(* Logix 5000 project; controller Receptivo vendor 1 type 14 code 106 rev 30.11; software revision 30.00; part 3 of 10 *)

   Impreso_3 : BOOL;
   Impreso_4 : BOOL;
   Imprimiendo_1 : BOOL;
   Imprimiendo_1_Timer : TIMER := (PRE := 7000);
   Imprimiendo_2 : BOOL;
   Imprimiendo_2_Timer : TIMER := (PRE := 7000);
   Imprimiendo_3 : BOOL;
   Imprimiendo_3_Timer : TIMER := (PRE := 7000);
   Imprimiendo_4 : BOOL;
   Imprimiendo_4_Timer : TIMER := (PRE := 7000);
   Index_Bidones_Videojet : DINT;
   Index_Elmar_Videojet : DINT := 112;
   Index_Fogg1_Videojet : DINT := 203;
   Index_Fogg2_Videojet : DINT := 23;
   Index_Karat_Videojet : DINT;
   Index_Karat_Videojet_Antiguo : DINT;
   Index_Productos : DINT := 118;
   Index_S : INT := 200;
   Index_Scanner : COUNTER := (PRE := 300, ACC := 3483, DN := 1);
   Indice_Bidon_Videojet : DINT;
   KEY_SWITCH_REM_RUN : BOOL := 1;
   KEY_SWITCH_RUN : BOOL;
   Latch_Scanner_1 : BOOL := 1;
   Latch_Scanner_2 : BOOL;
   Latch_Scanner_3 : BOOL;
   Lectura_Efectuada : BOOL;
   Linea_1 : SINT;
   Linea_2 : SINT;
   Linea_3 : SINT;
   Linea_4 : SINT;
   Linea_5 : SINT;
   Linea_General : SINT;
   LInea_General_1 : INT := 3;
   LInea_General_2 : INT := 1;
   LInea_General_3 : INT := 3;
   LInea_General_4 : INT := 5;
   Linea_String_General : STRING := '5';
   Listado : INT := 9;
   Listado_A : INT := 9;
   Lote : DINT := 148;
   Mes_dias : INT[13] := ([2] := 31, [3] := 59, [4] := 90, [5] := 120, [6] := 151, [7] := 181, [8] := 212, [9] := 243, [10] := 273, [11] := 304, [12] := 334);
   MODULE_FAULT_STATUS : DINT[10];
   Modulo_Ethernet_Mal : BOOL;
   new_day : BOOL;
   No_CAJAS_1 : DINT;
   No_CAJAS_2 : DINT;
   No_CAJAS_3 : DINT;
   No_existe : Descripcion := 'Codigo No Existe En El Inventario';
   Nuevo_Lote_Fogg1 : BOOL;
   Num_Cajas_Reales_1 : DINT;
   Num_Cajas_Reales_2 : DINT;
   Num_Cajas_Reales_3 : DINT;
   Num_Cajas_Reales_4 : DINT;
   Numero_Datos : DINT := 300;
   ons_add : BOOL;
   ons_add2 : BOOL;
   ons_add3 : BOOL;
   ons_add4 : BOOL;
   Ons_Cola2 : BOOL;
   Ons_Cola3 : BOOL;
   Ons_Corte_Dia : BOOL;
   ons_datos_mal_Bidones : BOOL;
   ons_datos_mal_elmar : BOOL;
   ons_datos_mal_Fogg1 : BOOL;
   ons_datos_mal_Fogg2 : BOOL;
   Ons_Datos_Mal_Karat : BOOL;
   ons_densidad_elmar : BOOL;
   ons_densidad_Fogg_1 : BOOL;
   Ons_Densidad_Karat : BOOL;
   Ons_NP : BOOL;
   Ons_NP2 : BOOL;
   Ons_NP3 : BOOL;
   Ons_NP4 : BOOL;
   Ons_Nuevo_Karat_Videojet : BOOL;
   ons_peso_caja_elmar_2 : BOOL;
   ONS_Reporte_Dia : BOOL;
   ons_scanner_1 : BOOL := 1;
   ons_scanner_3 : BOOL;
   ons_tare_station_4 : BOOL;
   Operador_1 : DINT := 5;
   Operador_2 : DINT := 5;
   Operador_3 : DINT := 5;
   Operador_4 : DINT := 6;
   PB_Enable_Scanner_1 : BOOL := 1;
   PB_Enable_Scanner_2 : BOOL;
   PB_Enable_Scanner_3 : BOOL;
   PB_Pesaje_1 : BOOL;
   PB_PV_Entre_Peso_Caja_Elmar : BOOL;
   PB_Tare_Station_1 : BOOL;
   PB_Tare_Station_2 : BOOL;
   PB_Tare_Station_3 : BOOL;
   PB_Tare_Station_4 : BOOL;
   Pesaje_1 : REAL := 0.6;
   Pesaje_2 : REAL := 0.6;
   Pesaje_3 : REAL := 0.9;
   Pesaje_4 : REAL := 0.102;
   Pesaje_Elmar_OK : BOOL;
   Pesaje_Fogg1_OK : BOOL;
   Pesaje_Fogg2_OK : BOOL;
   Pesaje_Karat_OK : BOOL;
   Peso_Aux : DINT;
   Peso_Aux_Scanner : STRING;
   Peso_Bidon : REAL;
   Peso_Bidones : REAL;
   Peso_Bidones_1 : REAL := 0.102;
   Peso_Caja_Bidones : REAL;
   Peso_Caja_Bidones_1 : REAL;
   Peso_Caja_Elmar : REAL;
   Peso_Caja_Elmar_1 : REAL := 0.6;
   Peso_Caja_Fogg1 : REAL;
   Peso_Caja_Fogg1_1 : REAL := 1.0;
   Peso_Caja_Fogg2 : REAL;
   Peso_Caja_Fogg2_1 : REAL := 0.9;
   Peso_Caja_Karat : REAL;
   Peso_Caja_Karat_1 : REAL;
   Peso_Mal_Estacion_1 : BOOL;
   Peso_Mal_Estacion_2 : BOOL;
   Peso_OK_Estacion_1 : BOOL;
   Peso_OK_Estacion_2 : BOOL;
   Peso_OK_Estacion_3 : BOOL;
   Peso_OK_Estacion_4 : BOOL;
   PESO_REAL_1 : DINT := -23;
   PESO_REAL_2 : DINT := -30;
   PESO_REAL_3 : DINT;
   PESO_REAL_4 : DINT := -23;
   PESO_TEORICO_1 : DINT := 865;
   PESO_TEORICO_2 : DINT := 585;
   PESO_TEORICO_3 : DINT := 865;
   PESO_TEORICO_4 : DINT := 786;
   Porcentaje_Peso_1 : REAL := 12257.143;
   Porcentaje_Peso_2 : REAL := 8257.143;
   Porcentaje_Peso_21 : DINT := 100;
   Porcentaje_Peso_3 : REAL := 10712.5;
   Porcentaje_Peso_4 : REAL := 1865.0;
   Print_1 : BOOL;
   Print_2 : BOOL;
   Print_3 : BOOL;
   Print_4 : BOOL;
   Printing_Enable : BOOL := 1;
   Producido_Bidones_Ahora : UDT_Maestro := (Descripcion := 'Dotchi Bidon x 20 L');
   Producido_Elmar_Ahora : UDT_Maestro := (Peso_Real_Estiba := 703.44, Peso_Teorico_Caja := 10.45, Codigo_EAN := '17702161409646', Codigo_QAD := '600620', Codigo_GCO := 600620, Descripcion := 'Alegria Caja 12 x 900 cm3  - Costa', Cajas_X_Estiba := 56, Codigo_Aceite := 600620, Envase := 900, Envases_x_Caja := 12);
   Producido_Fogg1_Ahora : UDT_Maestro := (Peso_Real_Estiba := 869.0, Peso_Teorico_Caja := 17.48, Codigo_EAN := '27702179003208', Codigo_QAD := '607490', Codigo_GCO := 607490, Descripcion := 'Vivi FF Caja 9 x2000 cm3 ', Cajas_X_Estiba := 42, Clima := 2, Codigo_Aceite := 607490, Envase := 2000, Envases_x_Caja := 9);
   Producido_Fogg2_Ahora : UDT_Maestro := (Peso_Real_Estiba := 691.2, Peso_Teorico_Caja := 17.3, Codigo_EAN := '17702161567070', Codigo_QAD := '605990', Codigo_GCO := 605990, Descripcion := 'Oriental 100% oleina x 3000 ML  Cj 6 Und', Cajas_X_Estiba := 50, Codigo_Aceite := 605990, Envase := 3000, Envases_x_Caja := 6);
   Producido_Karat_Ahora : UDT_Maestro;
   Producto1 : UDT_Inventario := (Peso_Teorico_Caja := 17.3, Descripcion := 'Oriental 100% ole$EDna x 3000 ML  Cj 6 Und', CajaXEstiba := 50, Codigo_Aceite := -1);
   Producto2 : UDT_Inventario := (Peso_Teorico_Caja := 10.45, Descripcion := 'Alegria Caja 12 x 900 cm3  - Costa', CajaXEstiba := 56, Codigo_Aceite := -1);
   Producto3 : UDT_Inventario := (Peso_Teorico_Caja := 17.3, Descripcion := 'Oriental 100% oleina x 3000 ML  Cj 6 Und', CajaXEstiba := 50, Codigo_Aceite := -1);
   Producto4 : UDT_Inventario := (Peso_Teorico_Caja := 16.38, Descripcion := 'Aceite Vegetal Torino  Exp.', CajaXEstiba := 48, Codigo_Aceite := -1);
   Producto_Codigo_Aceite_1 : DINT := -1;
   Producto_Codigo_Aceite_2 : DINT := -1;
   Producto_Codigo_Aceite_3 : DINT := -1;
   Producto_Codigo_Aceite_4 : DINT := -1;
   Producto_Scanner_1 : UDT_QAD;
   Producto_Scanner_11 : UDT_EAN14;
   Productos : UDT_Maestro[300] := ([0].Peso_Real_Estiba := 634.88, [0].Peso_Teorico_Caja := 14.72, [0].Codigo_EAN := '77702161305087', [0].Codigo_QAD := '600130', [0].Codigo_GCO := 600130, [0].Descripcion := 'Alegria Bidon x 15 L', [0].Cajas_X_Estiba := 48, [0].Clima := 2, [0].Codigo_Aceite := 600130, [0].Envase := 15000, [0].Envases_x_Caja := 1, [1].Peso_Real_Estiba := 690.84, [1].Peso_Teorico_Caja := 18.95, [1].Codigo_EAN := '07702161500506', [1].Codigo_QAD := '600100', [1].Codigo_GCO := 600100, [1].Descripcion := 'Alegria Bidon x 20 L', [1].Cajas_X_Estiba := 48, [1].Clima := 2, [1].Codigo_Aceite := 600100, [1].Envase := 20000, [1].Envases_x_Caja := 1, [2].Peso_Real_Estiba := 731.5, [2].Peso_Teorico_Caja := 18.8, [2].Codigo_EAN := '17702161574078', [2].Codigo_QAD := '606890', [2].Codigo_GCO := 606890, [2].Descripcion := 'Vivi FF Bidon x 20 L ', [2].Cajas_X_Estiba := 48, [2].Clima := 2, [2].Codigo_Aceite := 606890, [2].Envase := 20000, [2].Envases_x_Caja := 1, [3].Peso_Real_Estiba := 622.56, [3].Peso_Teorico_Caja := 19.31, [3].Codigo_EAN := '17702161071010', [3].Codigo_QAD := '606980', [3].Codigo_GCO := 606980, [3].Descripcion := 'Vivi FF Caja 4 x 5000 cm3 ', [3].Cajas_X_Estiba := 36, [3].Clima := 2, [3].Codigo_Aceite := 606980, [3].Envase := 5000, [3].Envases_x_Caja := 4, [4].Peso_Real_Estiba := 878.0, [4].Peso_Teorico_Caja := 17.4, [4].Codigo_EAN := '17702161987403', [4].Codigo_QAD := '607280', [4].Codigo_GCO := 607280, [4].Descripcion := 'Vivi FF Caja 6 x 3000 cm3 ', [4].Cajas_X_Estiba := 50, [4].Clima := 2, [4].Codigo_Aceite := 607280, [4].Envase := 3000, [4].Envases_x_Caja := 6, [5].Peso_Real_Estiba := 636.24, [5].Peso_Teorico_Caja := 17.54, [5].Codigo_EAN := '17702161845956', [5].Codigo_QAD := '607490', [5].Codigo_GCO := 607490,
        [5].Descripcion := 'Vivi FF Caja 9 x2000 cm3 ', [5].Cajas_X_Estiba := 42, [5].Clima := 2, [5].Codigo_Aceite := 607490, [5].Envase := 2000, [5].Envases_x_Caja := 9, [6].Peso_Real_Estiba := 627.2, [6].Peso_Teorico_Caja := 11.69, [6].Codigo_EAN := '17702161585364', [6].Codigo_QAD := '607690', [6].Codigo_GCO := 607690, [6].Descripcion := 'Vivi FF Caja 12 x 1000 cm3 ', [6].Cajas_X_Estiba := 70, [6].Clima := 2, [6].Codigo_Aceite := 607690, [6].Envase := 1000, [6].Envases_x_Caja := 12, [7].Peso_Real_Estiba := 830.0, [7].Peso_Teorico_Caja := 10.57, [7].Codigo_EAN := '17702161701764', [7].Codigo_QAD := '607890', [7].Codigo_GCO := 607890, [7].Descripcion := 'Vivi FF Caja 12 x 900 cm3 ', [7].Cajas_X_Estiba := 70, [7].Clima := 2, [7].Codigo_Aceite := 607890, [7].Envase := 900, [7].Envases_x_Caja := 12, [8].Peso_Real_Estiba := 625.1, [8].Peso_Teorico_Caja := 11.79, [8].Codigo_EAN := '17702161377068', [8].Codigo_QAD := '608090', [8].Codigo_GCO := 608090, [8].Descripcion := 'Vivi FF Caja 24 x 500 cm3 ', [8].Cajas_X_Estiba := 70, [8].Clima := 2, [8].Codigo_Aceite := 608090, [8].Envase := 500, [8].Envases_x_Caja := 24, [9].Peso_Real_Estiba := 770.0, [9].Peso_Teorico_Caja := 6.06, [9].Codigo_EAN := '17702161560002', [9].Codigo_QAD := '608290', [9].Codigo_GCO := 608290, [9].Descripcion := 'Vivi FF Caja 24 x 250 cm3 ', [9].Cajas_X_Estiba := 104, [9].Clima := 2, [9].Codigo_Aceite := 608290, [9].Envase := 250, [9].Envases_x_Caja := 24, [10].Peso_Real_Estiba := 883.2, [10].Peso_Teorico_Caja := 15.32, [10].Codigo_EAN := '67702179051603', [10].Codigo_QAD := '606280', [10].Codigo_GCO := 606280, [10].Descripcion := 'Comisariato Grasco Caja 6 x 2625 cm3', [10].Cajas_X_Estiba := 50, [10].Clima := 2, [10].Codigo_Aceite := 606280, [10].Envase := 2625,
        [10].Envases_x_Caja := 6, [11].Peso_Real_Estiba := 819.0, [11].Peso_Teorico_Caja := 17.27, [11].Codigo_EAN := '11111111111111', [11].Codigo_QAD := '602800', [11].Codigo_GCO := 602800, [11].Descripcion := 'La Muneca Comisariato Caja 6 x 3000 cm3', [11].Cajas_X_Estiba := 20, [11].Codigo_Aceite := 602800, [11].Envase := 3000, [11].Envases_x_Caja := 6, [12].Peso_Real_Estiba := 902.4, [12].Peso_Teorico_Caja := 19.44, [12].Codigo_EAN := '17702161301063', [12].Codigo_QAD := '601610', [12].Codigo_GCO := 601610, [12].Descripcion := 'Girasol de Oro Caja 4 x 5000 cm3', [12].Cajas_X_Estiba := 36, [12].Clima := 2, [12].Codigo_Aceite := 601610, [12].Envase := 5000, [12].Envases_x_Caja := 4, [13].Peso_Real_Estiba := 903.36, [13].Peso_Teorico_Caja := 17.47, [13].Codigo_EAN := '17702161301117', [13].Codigo_QAD := '601710', [13].Codigo_GCO := 601710, [13].Descripcion := 'Girasol de Oro Caja 6 x 3000 cm3', [13].Cajas_X_Estiba := 50, [13].Clima := 2, [13].Codigo_Aceite := 601710, [13].Envase := 3000, [13].Envases_x_Caja := 6, [14].Peso_Real_Estiba := 738.5, [14].Peso_Teorico_Caja := 17.57, [14].Codigo_EAN := '27702161301213', [14].Codigo_QAD := '601800', [14].Codigo_GCO := 601800, [14].Descripcion := 'Girasol de Oro Caja 9 x 2000 cm3', [14].Cajas_X_Estiba := 42, [14].Clima := 2, [14].Codigo_Aceite := 601800, [14].Envase := 2000, [14].Envases_x_Caja := 9, [15].Peso_Real_Estiba := 707.0, [15].Peso_Teorico_Caja := 11.69, [15].Codigo_EAN := '17702161301223', [15].Codigo_QAD := '601860', [15].Codigo_GCO := 601860, [15].Descripcion := 'Girasol de Oro Caja 12 x 1000 cm3', [15].Cajas_X_Estiba := 70, [15].Clima := 2, [15].Codigo_Aceite := 601860, [15].Envase := 1000, [15].Envases_x_Caja := 12, [16].Peso_Real_Estiba := 737.52, [16].Peso_Teorico_Caja := 11.83, [16].Codigo_EAN := '17702161301315', [16].Codigo_QAD := '602030', [16].Codigo_GCO := 602030,
        [16].Descripcion := 'Girasol de Oro$A0 Caja 24 x 500 cm3', [16].Cajas_X_Estiba := 70, [16].Clima := 2, [16].Codigo_Aceite := 602030, [16].Envase := 500, [16].Envases_x_Caja := 24, [17].Peso_Real_Estiba := 732.9, [17].Peso_Teorico_Caja := 18.89, [17].Codigo_EAN := '77702161302000', [17].Codigo_QAD := '604650', [17].Codigo_GCO := 604650, [17].Descripcion := 'Mazorca de oro Bidon x 20 L', [17].Cajas_X_Estiba := 48, [17].Clima := 2, [17].Codigo_Aceite := 604650, [17].Envase := 20000, [17].Envases_x_Caja := 1, [18].Peso_Real_Estiba := 731.22, [18].Peso_Teorico_Caja := 19.42, [18].Codigo_EAN := '17702161302107', [18].Codigo_QAD := '604750', [18].Codigo_GCO := 604750, [18].Descripcion := 'Mazorca de Oro caja 4 x 5000 cm3', [18].Cajas_X_Estiba := 36, [18].Clima := 2, [18].Codigo_Aceite := 604750, [18].Envase := 5000, [18].Envases_x_Caja := 4, [19].Peso_Real_Estiba := 869.0, [19].Peso_Teorico_Caja := 17.5, [19].Codigo_EAN := '17702161302152', [19].Codigo_QAD := '604850', [19].Codigo_GCO := 604850, [19].Descripcion := 'Mazorca de Oro Caja 6 x 3000 cm3', [19].Cajas_X_Estiba := 50, [19].Clima := 2, [19].Codigo_Aceite := 604850, [19].Envase := 3000, [19].Envases_x_Caja := 6, [20].Peso_Real_Estiba := 866.5, [20].Peso_Teorico_Caja := 17.57, [20].Codigo_EAN := '17702161302206', [20].Codigo_QAD := '605000', [20].Codigo_GCO := 605000, [20].Descripcion := 'Mazorca de Oro Caja 9 x 2000 cm3', [20].Cajas_X_Estiba := 42, [20].Clima := 2, [20].Codigo_Aceite := 605000, [20].Envase := 2000, [20].Envases_x_Caja := 9, [21].Peso_Real_Estiba := 871.0, [21].Peso_Teorico_Caja := 11.72, [21].Codigo_EAN := '17702161302251', [21].Codigo_QAD := '605150', [21].Codigo_GCO := 605150, [21].Descripcion := 'Mazorca de Oro Caja 12 x 1000 cm3', [21].Cajas_X_Estiba := 70, [21].Clima := 2, [21].Codigo_Aceite := 605150, [21].Envase := 1000,
        [21].Envases_x_Caja := 12, [22].Peso_Real_Estiba := 875.0, [22].Peso_Teorico_Caja := 11.83, [22].Codigo_EAN := '17702161302350', [22].Codigo_QAD := '605450', [22].Codigo_GCO := 605450, [22].Descripcion := 'Mazorca de Oro Caja 24 x 500 cm3', [22].Cajas_X_Estiba := 70, [22].Clima := 2, [22].Codigo_Aceite := 605450, [22].Envase := 500, [22].Envases_x_Caja := 24, [23].Peso_Real_Estiba := 691.2, [23].Peso_Teorico_Caja := 17.3, [23].Codigo_EAN := '17702161567070', [23].Codigo_QAD := '605990', [23].Codigo_GCO := 605990, [23].Descripcion := 'Oriental 100% oleina x 3000 ML  Cj 6 Und', [23].Cajas_X_Estiba := 50, [23].Codigo_Aceite := 605990, [23].Envase := 3000, [23].Envases_x_Caja := 6, [24].Peso_Real_Estiba := 690.48, [24].Peso_Teorico_Caja := 11.59, [24].Codigo_EAN := '17702161614989', [24].Codigo_QAD := '606180', [24].Codigo_GCO := 606180, [24].Descripcion := 'Oriental 100% oleina x 1000 ML Cj 12 Un', [24].Cajas_X_Estiba := 70, [24].Codigo_Aceite := 606180, [24].Envase := 1000, [24].Envases_x_Caja := 12, [25].Peso_Real_Estiba := 692.28, [25].Codigo_EAN := '17702161819711', [25].Codigo_QAD := '603240', [25].Codigo_GCO := 603240, [25].Descripcion := 'La Muneca 100% Oleina x 900 Ml', [25].Cajas_X_Estiba := 70, [25].Codigo_Aceite := 603240, [25].Envase := 900, [25].Envases_x_Caja := 12, [26].Peso_Real_Estiba := 823.2, [26].Codigo_EAN := '17702161540899', [26].Codigo_QAD := '603040', [26].Codigo_GCO := 603040, [26].Descripcion := 'La Muneca 100% Oleina x 1000 Ml', [26].Cajas_X_Estiba := 70, [26].Codigo_Aceite := 603040, [26].Envase := 1000, [26].Envases_x_Caja := 12, [27].Peso_Real_Estiba := 821.1, [27].Peso_Teorico_Caja := 18.73, [27].Codigo_EAN := '17702161816611', [27].Codigo_QAD := '606850', [27].Codigo_GCO := 606850, [27].Descripcion := 'Vivi 100% Oleina Bidon 20 L', [27].Cajas_X_Estiba := 48, [27].Codigo_Aceite := 606850, [27].Envase := 20000, [27].Envases_x_Caja := 1,
        [28].Peso_Real_Estiba := 819.0, [28].Peso_Teorico_Caja := 17.3, [28].Codigo_EAN := '17702161861642', [28].Codigo_QAD := '607180', [28].Codigo_GCO := 607180, [28].Descripcion := 'Vivi 100% Oleina Caja 6 x 3000 cm3 ', [28].Cajas_X_Estiba := 50, [28].Codigo_Aceite := 607180, [28].Envase := 3000, [28].Envases_x_Caja := 6, [29].Peso_Real_Estiba := 630.24, [29].Peso_Teorico_Caja := 11.59, [29].Codigo_EAN := '17702161372070', [29].Codigo_QAD := '607590', [29].Codigo_GCO := 607590, [29].Descripcion := 'Vivi 100% Oleina Caja 12 x 1000 cm3 ', [29].Cajas_X_Estiba := 70, [29].Codigo_Aceite := 607590, [29].Envase := 1000, [29].Envases_x_Caja := 12, [30].Peso_Real_Estiba := 629.2, [30].Peso_Teorico_Caja := 10.45, [30].Codigo_EAN := '17702161264023', [30].Codigo_QAD := '607790', [30].Codigo_GCO := 607790, [30].Descripcion := 'Vivi 100% Oleina  Caja 12 x 900 cm3 ', [30].Cajas_X_Estiba := 70, [30].Codigo_Aceite := 607790, [30].Envase := 900, [30].Envases_x_Caja := 12, [31].Peso_Real_Estiba := 630.24, [31].Peso_Teorico_Caja := 11.7, [31].Codigo_EAN := '17702161546570', [31].Codigo_QAD := '607990', [31].Codigo_GCO := 607990, [31].Descripcion := 'Vivi 100% Oleina Caja 24 x 500 cm3 ', [31].Cajas_X_Estiba := 70, [31].Codigo_Aceite := 607990, [31].Envase := 500, [31].Envases_x_Caja := 24, [32].Peso_Real_Estiba := 735.0, [32].Peso_Teorico_Caja := 19.18, [32].Codigo_EAN := '17702161071010', [32].Codigo_QAD := '607030', [32].Codigo_GCO := 607030, [32].Descripcion := 'Vivi F Caja 4 x 5000 cm3 ', [32].Cajas_X_Estiba := 36, [32].Clima := 1, [32].Codigo_Aceite := 607030, [32].Envase := 5000, [32].Envases_x_Caja := 4, [33].Peso_Real_Estiba := 735.0, [33].Peso_Teorico_Caja := 17.4, [33].Codigo_EAN := '17702161987403', [33].Codigo_QAD := '607230', [33].Codigo_GCO := 607230, [33].Descripcion := 'Vivi F Caja 6 x 3000 cm3 ', [33].Cajas_X_Estiba := 50, [33].Clima := 1, [33].Codigo_Aceite := 607230,
        [33].Envase := 3000, [33].Envases_x_Caja := 6, [34].Peso_Real_Estiba := 735.0, [34].Peso_Teorico_Caja := 17.45, [34].Codigo_EAN := '17702161845956', [34].Codigo_QAD := '607440', [34].Codigo_GCO := 607440, [34].Descripcion := 'Vivi F Caja 9 x2000 cm3 ', [34].Cajas_X_Estiba := 42, [34].Clima := 1, [34].Codigo_Aceite := 607440, [34].Envase := 2000, [34].Envases_x_Caja := 9, [35].Peso_Real_Estiba := 818.3, [35].Peso_Teorico_Caja := 11.63, [35].Codigo_EAN := '17702161585364', [35].Codigo_QAD := '607640', [35].Codigo_GCO := 607640, [35].Descripcion := 'Vivi F Caja 12 x 1000 cm3 ', [35].Cajas_X_Estiba := 70, [35].Clima := 1, [35].Codigo_Aceite := 607640, [35].Envase := 1000, [35].Envases_x_Caja := 12, [36].Peso_Real_Estiba := 814.8, [36].Peso_Teorico_Caja := 10.57, [36].Codigo_EAN := '17702161701764', [36].Codigo_QAD := '607840', [36].Codigo_GCO := 607890, [36].Descripcion := 'Vivi F Caja 12 x 900 cm3 ', [36].Cajas_X_Estiba := 70, [36].Clima := 2, [36].Codigo_Aceite := 607840, [36].Envase := 900, [36].Envases_x_Caja := 12, [37].Peso_Real_Estiba := 818.3, [37].Peso_Teorico_Caja := 11.73, [37].Codigo_EAN := '17702161377068', [37].Codigo_QAD := '608040', [37].Codigo_GCO := 608040, [37].Descripcion := 'Vivi F Caja 24 x 500 cm3 ', [37].Cajas_X_Estiba := 70, [37].Clima := 1, [37].Codigo_Aceite := 608040, [37].Envase := 500, [37].Envases_x_Caja := 24, [38].Peso_Real_Estiba := 907.2, [38].Peso_Teorico_Caja := 6.05, [38].Codigo_EAN := '17702161560002', [38].Codigo_QAD := '608240', [38].Codigo_GCO := 608240, [38].Descripcion := 'Vivi F Caja 24 x 250 cm3 ', [38].Cajas_X_Estiba := 104, [38].Clima := 1, [38].Codigo_Aceite := 608240, [38].Envase := 250, [38].Envases_x_Caja := 24, [39].Peso_Real_Estiba := 902.4, [39].Peso_Teorico_Caja := 18.74, [39].Codigo_QAD := '602360',
        [39].Codigo_GCO := 602360, [39].Descripcion := 'La Muneca Bidon x 20 L', [39].Cajas_X_Estiba := 48, [39].Codigo_Aceite := 602360, [39].Envase := 20000, [39].Envases_x_Caja := 1, [40].Peso_Real_Estiba := 902.4, [40].Peso_Teorico_Caja := 18.8, [40].Codigo_QAD := '602380', [40].Codigo_GCO := 602380, [40].Descripcion := 'La Muneca Bidon x 20 L ', [40].Cajas_X_Estiba := 48, [40].Clima := 2, [40].Codigo_Aceite := 602380, [40].Envase := 20000, [40].Envases_x_Caja := 1, [41].Peso_Real_Estiba := 737.8, [41].Peso_Teorico_Caja := 19.16, [41].Codigo_QAD := '602480', [41].Codigo_GCO := 602480, [41].Descripcion := 'La Muneca C Caja 4 x 5000 cm3 ', [41].Cajas_X_Estiba := 36, [41].Codigo_Aceite := 602480, [41].Envase := 5000, [41].Envases_x_Caja := 4, [42].Peso_Real_Estiba := 743.4, [42].Peso_Teorico_Caja := 17.26, [42].Codigo_QAD := '602680', [42].Codigo_GCO := 602680, [42].Descripcion := 'La Muneca C Caja 6 x 3000 cm3 ', [42].Cajas_X_Estiba := 50, [42].Codigo_Aceite := 602680, [42].Envase := 3000, [42].Envases_x_Caja := 6, [43].Peso_Real_Estiba := 824.6, [43].Peso_Teorico_Caja := 17.42, [43].Codigo_QAD := '602840', [43].Codigo_GCO := 602840, [43].Descripcion := 'La Muneca C Caja 9 x 2000 cm3 ', [43].Cajas_X_Estiba := 42, [43].Codigo_Aceite := 602840, [43].Envase := 2000, [43].Envases_x_Caja := 9, [44].Peso_Real_Estiba := 642.72, [44].Peso_Teorico_Caja := 11.63, [44].Codigo_QAD := '603040', [44].Codigo_GCO := 603040, [44].Descripcion := 'La Muneca  C Caja 12 x 1000 cm3 ', [44].Cajas_X_Estiba := 70, [44].Codigo_Aceite := 603040, [44].Envase := 1000, [44].Envases_x_Caja := 12, [45].Peso_Real_Estiba := 907.2, [45].Peso_Teorico_Caja := 10.46, [45].Codigo_QAD := '603240', [45].Codigo_GCO := 603240, [45].Descripcion := 'La Muneca C Caja 12 x 900 cm3 ', [45].Cajas_X_Estiba := 70, [45].Codigo_Aceite := 603240, [45].Envase := 900,
        [45].Envases_x_Caja := 12, [46].Peso_Real_Estiba := 693.72, [46].Peso_Teorico_Caja := 11.7, [46].Codigo_QAD := '603440', [46].Codigo_GCO := 603440, [46].Descripcion := 'La Muneca C Caja 24 x 500 cm3 ', [46].Cajas_X_Estiba := 70, [46].Codigo_Aceite := 603440, [46].Envase := 500, [46].Envases_x_Caja := 24, [47].Peso_Real_Estiba := 870.0, [47].Peso_Teorico_Caja := 6.06, [47].Codigo_QAD := '603640', [47].Codigo_GCO := 603640, [47].Descripcion := 'La Muneca C Caja 24 x 250 cm3 ', [47].Cajas_X_Estiba := 104, [47].Codigo_Aceite := 603640, [47].Envase := 250, [47].Envases_x_Caja := 24, [48].Peso_Real_Estiba := 830.2, [48].Peso_Teorico_Caja := 19.2, [48].Codigo_QAD := '602530', [48].Codigo_GCO := 602530, [48].Descripcion := 'La Muneca F Caja 4 x 5000 cm3 ', [48].Cajas_X_Estiba := 36, [48].Clima := 1, [48].Codigo_Aceite := 602530, [48].Envase := 5000, [48].Envases_x_Caja := 4, [49].Peso_Real_Estiba := 632.32, [49].Peso_Teorico_Caja := 17.33, [49].Codigo_EAN := '17702161143267', [49].Codigo_QAD := '602740', [49].Codigo_GCO := 602740, [49].Descripcion := 'La Muneca F Caja 6 x 3000 cm3 ', [49].Cajas_X_Estiba := 50, [49].Clima := 1, [49].Codigo_Aceite := 602740, [49].Envase := 3000, [49].Envases_x_Caja := 6, [50].Peso_Real_Estiba := 728.7, [50].Peso_Teorico_Caja := 17.45, [50].Codigo_QAD := '602890', [50].Codigo_GCO := 602890, [50].Descripcion := 'La Muneca F Caja 9 x 2000 cm3 ', [50].Cajas_X_Estiba := 42, [50].Clima := 1, [50].Codigo_Aceite := 602890, [50].Envase := 2000, [50].Envases_x_Caja := 9, [51].Peso_Real_Estiba := 743.4, [51].Peso_Teorico_Caja := 10.48, [51].Codigo_EAN := '17702161422836', [51].Codigo_QAD := '603090', [51].Codigo_GCO := 603290, [51].Descripcion := 'La Muneca F Caja 12 x 900 cm3 ', [51].Cajas_X_Estiba := 70, [51].Clima := 1, [51].Codigo_Aceite := 603090, [51].Envase := 900,
        [51].Envases_x_Caja := 12, [52].Peso_Real_Estiba := 821.1, [52].Peso_Teorico_Caja := 11.73, [52].Codigo_QAD := '603490', [52].Codigo_GCO := 603490, [52].Descripcion := 'La Muneca F Caja 24 x 500 cm3 ', [52].Cajas_X_Estiba := 70, [52].Clima := 1, [52].Codigo_Aceite := 603490, [52].Envase := 500, [52].Envases_x_Caja := 24, [53].Peso_Real_Estiba := 875.0, [53].Peso_Teorico_Caja := 6.05, [53].Codigo_QAD := '603690', [53].Codigo_GCO := 603690, [53].Descripcion := 'La Muneca F Caja 24 x 250 cm3 ', [53].Cajas_X_Estiba := 104, [53].Clima := 1, [53].Codigo_Aceite := 603690, [53].Envase := 250, [53].Envases_x_Caja := 24, [54].Peso_Real_Estiba := 698.4, [54].Peso_Teorico_Caja := 19.3, [54].Codigo_QAD := '602580', [54].Codigo_GCO := 602580, [54].Descripcion := 'La Muneca FF Caja 4 x 5000 cm3 ', [54].Cajas_X_Estiba := 36, [54].Clima := 2, [54].Codigo_Aceite := 602580, [54].Envase := 5000, [54].Envases_x_Caja := 4, [55].Peso_Real_Estiba := 746.9, [55].Peso_Teorico_Caja := 17.37, [55].Codigo_QAD := '602790', [55].Codigo_GCO := 602790, [55].Descripcion := 'La Muneca FF Caja 6 x 3000 cm3 ', [55].Cajas_X_Estiba := 50, [55].Clima := 2, [55].Codigo_Aceite := 602790, [55].Envase := 3000, [55].Envases_x_Caja := 6, [56].Peso_Real_Estiba := 908.16, [56].Peso_Teorico_Caja := 17.48, [56].Codigo_EAN := '17702161885983', [56].Codigo_QAD := '602940', [56].Codigo_GCO := 602940, [56].Descripcion := 'La Muneca FF Caja 9 x 2000 cm3 ', [56].Cajas_X_Estiba := 42, [56].Clima := 2, [56].Codigo_Aceite := 602940, [56].Envase := 2000, [56].Envases_x_Caja := 9, [57].Peso_Real_Estiba := 634.128, [57].Peso_Teorico_Caja := 11.65, [57].Codigo_QAD := '603140', [57].Codigo_GCO := 603140, [57].Descripcion := 'La Muneca FF Caja 12 x 1000 cm3 ', [57].Cajas_X_Estiba := 70, [57].Clima := 2, [57].Codigo_Aceite := 603140,
        [57].Envase := 1000, [57].Envases_x_Caja := 12, [58].Peso_Real_Estiba := 743.4, [58].Peso_Teorico_Caja := 10.54, [58].Codigo_QAD := '603340', [58].Codigo_GCO := 603340, [58].Descripcion := 'La Muneca FF Caja 12 x 900 cm3 ', [58].Cajas_X_Estiba := 70, [58].Clima := 2, [58].Codigo_Aceite := 603340, [58].Envase := 900, [58].Envases_x_Caja := 12, [59].Peso_Real_Estiba := 831.5, [59].Peso_Teorico_Caja := 11.73, [59].Codigo_QAD := '603540', [59].Codigo_GCO := 603540, [59].Descripcion := 'La Muneca  FF Caja 24 x 500 cm3 ', [59].Cajas_X_Estiba := 70, [59].Clima := 2, [59].Codigo_Aceite := 603540, [59].Envase := 500, [59].Envases_x_Caja := 24, [60].Peso_Real_Estiba := 698.4, [60].Peso_Teorico_Caja := 6.06, [60].Codigo_QAD := '603740', [60].Codigo_GCO := 603740, [60].Descripcion := 'La Muneca FF Caja 24 x 250 cm3 ', [60].Cajas_X_Estiba := 104, [60].Clima := 2, [60].Codigo_Aceite := 603740, [60].Envase := 250, [60].Envases_x_Caja := 24, [61].Peso_Real_Estiba := 829.5, [61].Peso_Teorico_Caja := 17.39, [61].Codigo_EAN := '07702179001033', [61].Codigo_QAD := '626510', [61].Codigo_GCO := 626510, [61].Descripcion := 'Sarita  Soya-palma Bidon x 18 L', [61].Cajas_X_Estiba := 48, [61].Codigo_Aceite := 626510, [61].Envase := 18000, [61].Envases_x_Caja := 1, [62].Peso_Real_Estiba := 742.7, [62].Peso_Teorico_Caja := 19.18, [62].Codigo_EAN := '06151710202004', [62].Codigo_QAD := '626550', [62].Codigo_GCO := 626550, [62].Descripcion := 'Sarita Soya-Palma  Caja 4 x 5000 cm3', [62].Cajas_X_Estiba := 36, [62].Codigo_Aceite := 626550, [62].Envase := 5000, [62].Envases_x_Caja := 4, [63].Peso_Real_Estiba := 875.0, [63].Peso_Teorico_Caja := 17.34, [63].Codigo_EAN := '67702179091408', [63].Codigo_QAD := '626800', [63].Codigo_GCO := 626800, [63].Descripcion := 'Sarita Soya-Palma Caja 6 x 3000 cm3', [63].Cajas_X_Estiba := 50, [63].Codigo_Aceite := 626800,
        [63].Envase := 3000, [63].Envases_x_Caja := 6, [64].Peso_Real_Estiba := 627.2, [64].Peso_Teorico_Caja := 12.84, [64].Codigo_EAN := '00001517101902', [64].Codigo_QAD := '626950', [64].Codigo_GCO := 626950, [64].Descripcion := 'Sarita Soya-Palma Caja 8 x 1600 cm3', [64].Cajas_X_Estiba := 48, [64].Codigo_Aceite := 626950, [64].Envase := 1600, [64].Envases_x_Caja := 8, [65].Peso_Real_Estiba := 739.2, [65].Peso_Teorico_Caja := 16.6, [65].Codigo_EAN := '67702179091507', [65].Codigo_QAD := '627130', [65].Codigo_GCO := 627130, [65].Descripcion := 'Sarita Soya-Palma Caja 12 x 1.4 cm3', [65].Cajas_X_Estiba := 50, [65].Codigo_Aceite := 627130, [65].Envase := 1400, [65].Envases_x_Caja := 12, [66].Peso_Real_Estiba := 826.0, [66].Peso_Teorico_Caja := 10.48, [66].Codigo_EAN := '67702179594704', [66].Codigo_QAD := '627200', [66].Codigo_GCO := 627200, [66].Descripcion := 'Sarita Soya-Palma Caja 12 x 900 cm3', [66].Cajas_X_Estiba := 70, [66].Codigo_Aceite := 627200, [66].Envase := 900, [66].Envases_x_Caja := 12, [67].Peso_Real_Estiba := 826.0, [67].Peso_Teorico_Caja := 8.83, [67].Codigo_EAN := '67702179091606', [67].Codigo_QAD := '627300', [67].Codigo_GCO := 627300, [67].Descripcion := 'Sarita Soya-Palma Caja 12 x 750 cm3', [67].Cajas_X_Estiba := 70, [67].Codigo_Aceite := 627300, [67].Envase := 750, [67].Envases_x_Caja := 12, [68].Peso_Real_Estiba := 636.48, [68].Peso_Teorico_Caja := 9.5, [68].Codigo_EAN := '67702179091705', [68].Codigo_QAD := '627500', [68].Codigo_GCO := 627500, [68].Descripcion := 'Sarita Soya-Palma Caja 24 x 400 cm3', [68].Cajas_X_Estiba := 66, [68].Codigo_Aceite := 627500, [68].Envase := 400, [68].Envases_x_Caja := 24, [69].Peso_Real_Estiba := 880.5, [69].Peso_Teorico_Caja := 4.9, [69].Codigo_EAN := '67702179091804', [69].Codigo_QAD := '627650', [69].Codigo_GCO := 627650, [69].Descripcion := 'Sarita Soya-Palma Caja 24 x 200 cm3', [69].Cajas_X_Estiba := 128, [69].Codigo_Aceite := 627650,
        [69].Envase := 200, [69].Envases_x_Caja := 24, [70].Peso_Real_Estiba := 746.9, [70].Peso_Teorico_Caja := 6.11, [70].Codigo_EAN := '17702109017766', [70].Codigo_QAD := '604310', [70].Codigo_GCO := 604310, [70].Descripcion := 'Sevillana caja 24 $A0x 250 cm3 ', [70].Cajas_X_Estiba := 78, [70].Clima := 2, [70].Codigo_Aceite := 604310, [70].Envase := 250, [70].Envases_x_Caja := 24, [71].Peso_Real_Estiba := 829.78, [71].Peso_Teorico_Caja := 11.85, [71].Codigo_EAN := '17702109017773', [71].Codigo_QAD := '604320', [71].Codigo_GCO := 604320, [71].Descripcion := 'Sevillana caja 24 x 500 cm3', [71].Cajas_X_Estiba := 40, [71].Clima := 2, [71].Codigo_Aceite := 604320, [71].Envase := 500, [71].Envases_x_Caja := 24, [72].Peso_Real_Estiba := 743.4, [72].Peso_Teorico_Caja := 10.55, [72].Codigo_EAN := '17702109017254', [72].Codigo_QAD := '604330', [72].Codigo_GCO := 604330, [72].Descripcion := 'Sevillana$A0caja 12 $A0x 900 cm3 ', [72].Cajas_X_Estiba := 56, [72].Clima := 2, [72].Codigo_Aceite := 604330, [72].Envase := 900, [72].Envases_x_Caja := 12, [73].Peso_Real_Estiba := 831.5, [73].Peso_Teorico_Caja := 11.72, [73].Codigo_EAN := '17702109017759', [73].Codigo_QAD := '604340', [73].Codigo_GCO := 604340, [73].Descripcion := 'Sevillana caja 12 x 1000 cm3', [73].Cajas_X_Estiba := 44, [73].Clima := 2, [73].Codigo_Aceite := 604340, [73].Envase := 1000, [73].Envases_x_Caja := 12, [74].Peso_Real_Estiba := 830.9, [74].Peso_Teorico_Caja := 17.5, [74].Codigo_EAN := '17702141064681', [74].Codigo_QAD := '604350', [74].Codigo_GCO := 604350, [74].Descripcion := 'Sevillana$A0caja 6 $A0x 3000 cm3', [74].Cajas_X_Estiba := 45, [74].Clima := 2, [74].Codigo_Aceite := 604350, [74].Envase := 3000, [74].Envases_x_Caja := 6, [75].Peso_Real_Estiba := 868.55, [75].Peso_Teorico_Caja := 17.5, [75].Codigo_EAN := '17702109000102',
        [75].Codigo_QAD := '604390', [75].Codigo_GCO := 604390, [75].Descripcion := 'Purisimo caja  6 x 3000 cm3', [75].Cajas_X_Estiba := 45, [75].Clima := 2, [75].Codigo_Aceite := 604390, [75].Envase := 3000, [75].Envases_x_Caja := 6, [76].Peso_Real_Estiba := 693.792, [76].Peso_Teorico_Caja := 11.72, [76].Codigo_EAN := '17702109000089', [76].Codigo_QAD := '604380', [76].Codigo_GCO := 604380, [76].Descripcion := 'Purisimo caja$A0 12 x 1000 cm3', [76].Cajas_X_Estiba := 44, [76].Clima := 2, [76].Codigo_Aceite := 604380, [76].Envase := 1000, [76].Envases_x_Caja := 12, [77].Peso_Real_Estiba := 640.2, [77].Peso_Teorico_Caja := 10.55, [77].Codigo_EAN := '17702109009525', [77].Codigo_QAD := '604370', [77].Codigo_GCO := 604370, [77].Descripcion := 'Purisimo$A0 caja 12 x 900 cm3', [77].Cajas_X_Estiba := 56, [77].Clima := 2, [77].Codigo_Aceite := 604370, [77].Envase := 900, [77].Envases_x_Caja := 12, [78].Peso_Real_Estiba := 629.76, [78].Peso_Teorico_Caja := 11.85, [78].Codigo_EAN := '17702109000065', [78].Codigo_QAD := '604360', [78].Codigo_GCO := 604360, [78].Descripcion := 'Purisimo  Caja 24  x 500 cm3 ', [78].Cajas_X_Estiba := 40, [78].Clima := 2, [78].Codigo_Aceite := 604360, [78].Envase := 500, [78].Envases_x_Caja := 24, [79].Peso_Real_Estiba := 619.776, [79].Peso_Teorico_Caja := 17.5, [79].Codigo_EAN := '17702141000252', [79].Codigo_QAD := '604430', [79].Codigo_GCO := 604430, [79].Descripcion := 'Z caja 6 x 3000 cm3', [79].Cajas_X_Estiba := 45, [79].Clima := 2, [79].Codigo_Aceite := 604430, [79].Envase := 3000, [79].Envases_x_Caja := 6, [80].Peso_Teorico_Caja := 11.72, [80].Codigo_EAN := '17702141000238', [80].Codigo_QAD := '604410', [80].Codigo_GCO := 604410, [80].Descripcion := 'Z  caja 12 x 1000 cm3', [80].Cajas_X_Estiba := 44, [80].Clima := 2, [80].Codigo_Aceite := 604410,
        [80].Envase := 1000, [80].Envases_x_Caja := 12, [81].Peso_Teorico_Caja := 11.85, [81].Codigo_EAN := '17702141000214', [81].Codigo_QAD := '604400', [81].Codigo_GCO := 604400, [81].Descripcion := 'Z caja$A0 24 x 500 cm3', [81].Cajas_X_Estiba := 40, [81].Clima := 2, [81].Codigo_Aceite := 604400, [81].Envase := 500, [81].Envases_x_Caja := 24, [82].Peso_Real_Estiba := 622.08, [82].Peso_Teorico_Caja := 10.55, [82].Codigo_EAN := '17702109009501', [82].Codigo_QAD := '604420', [82].Codigo_GCO := 604420, [82].Descripcion := 'Z caja 12 x 900 cm3', [82].Cajas_X_Estiba := 56, [82].Clima := 2, [82].Codigo_Aceite := 604420, [82].Envase := 900, [82].Envases_x_Caja := 12, [83].Peso_Real_Estiba := 877.0, [83].Peso_Teorico_Caja := 17.5, [83].Codigo_EAN := '17702109019739', [83].Codigo_QAD := '604470', [83].Codigo_GCO := 604470, [83].Descripcion := 'Mallorca caja 6x3000 cm3', [83].Cajas_X_Estiba := 45, [83].Clima := 2, [83].Codigo_Aceite := 604470, [83].Envase := 3000, [83].Envases_x_Caja := 6, [84].Peso_Real_Estiba := 689.184, [84].Peso_Teorico_Caja := 11.72, [84].Codigo_EAN := '17702109019692', [84].Codigo_QAD := '604460', [84].Codigo_GCO := 604460, [84].Descripcion := 'Mallorca$A0 caja 12x1000$A0 cm3', [84].Cajas_X_Estiba := 44, [84].Clima := 2, [84].Codigo_Aceite := 604460, [84].Envase := 1000, [84].Envases_x_Caja := 12, [85].Peso_Real_Estiba := 637.56, [85].Peso_Teorico_Caja := 10.55, [85].Codigo_EAN := '17702109019685', [85].Codigo_QAD := '604450', [85].Codigo_GCO := 604450, [85].Descripcion := 'Mallorca caja 12x900 cm3', [85].Cajas_X_Estiba := 56, [85].Clima := 2, [85].Codigo_Aceite := 604450, [85].Envase := 900, [85].Envases_x_Caja := 12, [86].Peso_Real_Estiba := 624.64, [86].Peso_Teorico_Caja := 11.85, [86].Codigo_EAN := '17702109019487', [86].Codigo_QAD := '604440',
        [86].Codigo_GCO := 604440, [86].Descripcion := 'Mallorca caja 24x500 cm3', [86].Cajas_X_Estiba := 40, [86].Clima := 2, [86].Codigo_Aceite := 604440, [86].Envase := 500, [86].Envases_x_Caja := 24, [87].Peso_Real_Estiba := 622.3, [87].Peso_Teorico_Caja := 17.5, [87].Codigo_EAN := '17702109009280', [87].Codigo_QAD := '604500', [87].Codigo_GCO := 604500, [87].Descripcion := 'Soy sabor caja$A0 6 x 3000cm3', [87].Cajas_X_Estiba := 45, [87].Clima := 2, [87].Codigo_Aceite := 604500, [87].Envase := 3000, [87].Envases_x_Caja := 6, [88].Peso_Real_Estiba := 619.99, [88].Peso_Teorico_Caja := 11.72, [88].Codigo_EAN := '17702109007958', [88].Codigo_QAD := '604480', [88].Codigo_GCO := 604480, [88].Descripcion := 'Soy sabor caja 12 x 1000 cm3', [88].Cajas_X_Estiba := 44, [88].Clima := 2, [88].Codigo_Aceite := 604480, [88].Envase := 1000, [88].Envases_x_Caja := 12, [89].Peso_Real_Estiba := 830.0, [89].Peso_Teorico_Caja := 10.55, [89].Codigo_EAN := '17702109009518', [89].Codigo_QAD := '604490', [89].Codigo_GCO := 604490, [89].Descripcion := 'Soy sabor caja$A0 12 x 900 cm3', [89].Cajas_X_Estiba := 56, [89].Clima := 2, [89].Codigo_Aceite := 604490, [89].Envase := 900, [89].Envases_x_Caja := 12, [90].Peso_Real_Estiba := 730.8, [90].Peso_Teorico_Caja := 17.4, [90].Codigo_EAN := '67702179504208', [90].Codigo_QAD := '629600', [90].Codigo_GCO := 629600, [90].Descripcion := 'Medalla de Oro 3000 cm$B3 Cj 6 Un', [90].Cajas_X_Estiba := 50, [90].Clima := 2, [90].Codigo_Aceite := 629600, [90].Envase := 3000, [90].Envases_x_Caja := 6, [91].Peso_Real_Estiba := 870.0, [91].Peso_Teorico_Caja := 19.18, [91].Codigo_EAN := '17705946722902', [91].Codigo_QAD := '634260', [91].Codigo_GCO := 634260, [91].Descripcion := 'Alkosto 6 x 5000 cm3', [91].Cajas_X_Estiba := 36, [91].Clima := 2, [91].Codigo_Aceite := 634260,
        [91].Envase := 5000, [91].Envases_x_Caja := 4, [92].Peso_Real_Estiba := 694.8, [92].Peso_Teorico_Caja := 17.5, [92].Codigo_EAN := '17705946722896', [92].Codigo_QAD := '634230', [92].Codigo_GCO := 634230, [92].Descripcion := 'Alkosto  6 x 3000 cm3', [92].Cajas_X_Estiba := 50, [92].Clima := 2, [92].Codigo_Aceite := 634230, [92].Envase := 3000, [92].Envases_x_Caja := 6, [93].Peso_Real_Estiba := 826.0, [93].Peso_Teorico_Caja := 11.69, [93].Codigo_EAN := '17705946722889', [93].Codigo_QAD := '634220', [93].Codigo_GCO := 634220, [93].Descripcion := 'Alkosto 12 x 1000 cm3', [93].Cajas_X_Estiba := 70, [93].Clima := 2, [93].Codigo_Aceite := 634220, [93].Envase := 1000, [93].Envases_x_Caja := 12, [94].Peso_Real_Estiba := 624.0, [94].Peso_Teorico_Caja := 18.8, [94].Codigo_EAN := '17705946722919', [94].Codigo_QAD := '634250', [94].Codigo_GCO := 634250, [94].Descripcion := 'Alkosto Bid$F3n 20 Lt', [94].Cajas_X_Estiba := 48, [94].Clima := 2, [94].Codigo_Aceite := 634250, [94].Envase := 20000, [94].Envases_x_Caja := 1, [95].Peso_Real_Estiba := 819.0, [95].Peso_Teorico_Caja := 17.5, [95].Codigo_EAN := '17705946719377', [95].Codigo_QAD := '634280', [95].Codigo_GCO := 634280, [95].Descripcion := 'MiDia 6 x 3000 cm3', [95].Cajas_X_Estiba := 50, [95].Clima := 2, [95].Codigo_Aceite := 634280, [95].Envase := 3000, [95].Envases_x_Caja := 6, [96].Peso_Real_Estiba := 921.6, [96].Peso_Teorico_Caja := 17.54, [96].Codigo_EAN := '17705946719391', [96].Codigo_QAD := '634240', [96].Codigo_GCO := 634240, [96].Descripcion := 'MiDia 9 x 2000 cm3', [96].Cajas_X_Estiba := 42, [96].Clima := 2, [96].Codigo_Aceite := 634240, [96].Envase := 2000, [96].Envases_x_Caja := 9, [97].Peso_Real_Estiba := 880.0, [97].Peso_Teorico_Caja := 11.69, [97].Codigo_EAN := '17705946719360',
        [97].Codigo_QAD := '634270', [97].Codigo_GCO := 634270, [97].Descripcion := 'MiDia 12 x 1000 cm3', [97].Cajas_X_Estiba := 70, [97].Clima := 2, [97].Codigo_Aceite := 634270, [97].Envase := 1000, [97].Envases_x_Caja := 12, [98].Peso_Real_Estiba := 827.4, [98].Peso_Teorico_Caja := 11.73, [98].Codigo_EAN := '17705946719384', [98].Codigo_QAD := '634210', [98].Codigo_GCO := 634210, [98].Descripcion := 'MiDia 24 x 500 cm3', [98].Cajas_X_Estiba := 70, [98].Clima := 1, [98].Codigo_Aceite := 634210, [98].Envase := 500, [98].Envases_x_Caja := 24, [99].Peso_Real_Estiba := 634.4, [99].Peso_Teorico_Caja := 18.95, [99].Codigo_EAN := '22222222222222', [99].Codigo_QAD := '600050', [99].Codigo_GCO := 600050, [99].Descripcion := 'Alegria 20Z x 20 LT', [99].Cajas_X_Estiba := 48, [99].Clima := 2, [99].Codigo_Aceite := 600050, [99].Envase := 20000, [99].Envases_x_Caja := 1, [100].Peso_Real_Estiba := 741.3, [100].Peso_Teorico_Caja := 18.8, [100].Codigo_EAN := '17702179010325', [100].Codigo_QAD := '590320', [100].Codigo_GCO := 590320, [100].Descripcion := 'Vivi SuperFreidor x 20 LT', [100].Cajas_X_Estiba := 48, [100].Clima := 2, [100].Codigo_Aceite := 590320, [100].Envase := 20000, [100].Envases_x_Caja := 1, [101].Peso_Real_Estiba := 820.4, [101].Peso_Teorico_Caja := 17.38, [101].Codigo_EAN := '17702161303159', [101].Codigo_QAD := '605950', [101].Codigo_GCO := 605950, [101].Descripcion := 'Oriental Mezcla Caja 6 x 3000 cm3', [101].Cajas_X_Estiba := 50, [101].Clima := 2, [101].Codigo_Aceite := 605950, [101].Envase := 3000, [101].Envases_x_Caja := 6, [102].Peso_Real_Estiba := 904.32, [102].Peso_Teorico_Caja := 11.67, [102].Codigo_EAN := '17702161303258', [102].Codigo_QAD := '606150', [102].Codigo_GCO := 606150, [102].Descripcion := 'Oriental Mezcla Caja 12 x 1000 cm3', [102].Cajas_X_Estiba := 70, [102].Clima := 2,
        [102].Codigo_Aceite := 606150, [102].Envase := 1000, [102].Envases_x_Caja := 12, [103].Peso_Real_Estiba := 875.0, [103].Peso_Teorico_Caja := 17.38, [103].Codigo_EAN := '67702179504208', [103].Codigo_QAD := '629600', [103].Codigo_GCO := 629600, [103].Descripcion := 'Medalla de Oro vegetal Caja 6 x 3000 cm3', [103].Cajas_X_Estiba := 50, [103].Clima := 2, [103].Codigo_Aceite := 629600, [103].Envase := 3000, [103].Envases_x_Caja := 6, [104].Peso_Real_Estiba := 875.0, [104].Peso_Teorico_Caja := 18.4, [104].Codigo_EAN := '07702179010332', [104].Codigo_QAD := '628250', [104].Codigo_GCO := 628250, [104].Descripcion := 'Soya RBD Bidon x 20 L', [104].Cajas_X_Estiba := 48, [104].Clima := 2, [104].Codigo_Aceite := 628250, [104].Envase := 20000, [104].Envases_x_Caja := 1, [105].Peso_Real_Estiba := 969.0, [105].Peso_Teorico_Caja := 10.45, [105].Codigo_EAN := '17702161264023', [105].Codigo_QAD := '590330', [105].Codigo_GCO := 590330, [105].Descripcion := 'Vivi Oleina 12 x 900   cm3 -Exp', [105].Cajas_X_Estiba := 70, [105].Codigo_Aceite := 590330, [105].Envase := 900, [105].Envases_x_Caja := 12, [106].Peso_Real_Estiba := 903.36, [106].Peso_Teorico_Caja := 17.3, [106].Codigo_EAN := '17705946789233', [106].Codigo_QAD := '634340', [106].Codigo_GCO := 634340, [106].Descripcion := 'Midia 6 x 3000 ml - Costa', [106].Cajas_X_Estiba := 50, [106].Codigo_Aceite := 634340, [106].Envase := 3000, [106].Envases_x_Caja := 6, [107].Peso_Real_Estiba := 875.0, [107].Peso_Teorico_Caja := 17.45, [107].Codigo_EAN := '17705946789226', [107].Codigo_QAD := '634330', [107].Codigo_GCO := 634330, [107].Descripcion := 'Midia 9 x 2000 ml - Costa', [107].Cajas_X_Estiba := 42, [107].Codigo_Aceite := 634330, [107].Envase := 2000, [107].Envases_x_Caja := 9, [108].Peso_Real_Estiba := 694.8, [108].Peso_Teorico_Caja := 11.59, [108].Codigo_EAN := '17705946789219', [108].Codigo_QAD := '634320', [108].Codigo_GCO := 634320,
        [108].Descripcion := 'Midia 12 x 1000 ml - Costa', [108].Cajas_X_Estiba := 70, [108].Codigo_Aceite := 634320, [108].Envase := 1000, [108].Envases_x_Caja := 12, [109].Peso_Real_Estiba := 739.2, [109].Peso_Teorico_Caja := 11.7, [109].Codigo_EAN := '17705946789202', [109].Codigo_QAD := '634310', [109].Codigo_GCO := 634310, [109].Descripcion := 'Midia 24 x 500 ml - Costa', [109].Cajas_X_Estiba := 70, [109].Codigo_Aceite := 634310, [109].Envase := 500, [109].Envases_x_Caja := 24, [110].Peso_Real_Estiba := 825.3, [110].Peso_Teorico_Caja := 17.38, [110].Codigo_EAN := '17702161501005', [110].Codigo_QAD := '600250', [110].Codigo_GCO := 600250, [110].Descripcion := 'Alegria Caja 6 x 3000 - Mezcla', [110].Cajas_X_Estiba := 30, [110].Clima := 2, [110].Codigo_Aceite := 600250, [110].Envase := 3000, [110].Envases_x_Caja := 6, [111].Peso_Real_Estiba := 875.0, [111].Peso_Teorico_Caja := 17.3, [111].Codigo_EAN := '17702161043987', [111].Codigo_QAD := '600300', [111].Codigo_GCO := 600300, [111].Descripcion := 'Alegria Caja 6 x 3000 cm3  - Costa', [111].Cajas_X_Estiba := 30, [111].Codigo_Aceite := 600300, [111].Envase := 3000, [111].Envases_x_Caja := 6, [112].Peso_Real_Estiba := 703.44, [112].Peso_Teorico_Caja := 10.45, [112].Codigo_EAN := '17702161409646', [112].Codigo_QAD := '600620', [112].Codigo_GCO := 600620, [112].Descripcion := 'Alegria Caja 12 x 900 cm3  - Costa', [112].Cajas_X_Estiba := 56, [112].Codigo_Aceite := 600620, [112].Envase := 900, [112].Envases_x_Caja := 12, [113].Peso_Real_Estiba := 819.0, [113].Peso_Teorico_Caja := 6.04, [113].Codigo_EAN := '67702179014202', [113].Codigo_QAD := '608190', [113].Codigo_GCO := 608190, [113].Descripcion := 'Vivi 100% Oleina Caja 24 x 250 cm3', [113].Cajas_X_Estiba := 104, [113].Codigo_Aceite := 608190, [113].Envase := 250, [113].Envases_x_Caja := 24, [114].Peso_Real_Estiba := 747.6, [114].Peso_Teorico_Caja := 16.77, [114].Codigo_EAN := '17702161075919', [114].Codigo_QAD := '606990',
        [114].Codigo_GCO := 606990, [114].Descripcion := 'Bidon 18 LT  - Export Panama', [114].Cajas_X_Estiba := 48, [114].Codigo_Aceite := 606990, [114].Envase := 18000, [114].Envases_x_Caja := 1, [115].Peso_Real_Estiba := 880.0, [115].Peso_Teorico_Caja := 16.77, [115].Codigo_EAN := '17702161411670', [115].Codigo_QAD := '607000', [115].Codigo_GCO := 607000, [115].Descripcion := 'Bidon 18 LT  - Export Falcon', [115].Cajas_X_Estiba := 48, [115].Codigo_Aceite := 607000, [115].Envase := 18000, [115].Envases_x_Caja := 1, [116].Peso_Real_Estiba := 698.4, [116].Peso_Teorico_Caja := 16.77, [116].Codigo_EAN := '17702161555343', [116].Codigo_QAD := '607010', [116].Codigo_GCO := 607010, [116].Descripcion := 'Aceite vegetal Lila 18 Lt  Exp', [116].Cajas_X_Estiba := 48, [116].Codigo_Aceite := 607010, [116].Envase := 18000, [116].Envases_x_Caja := 1, [117].Peso_Real_Estiba := 828.8, [117].Peso_Teorico_Caja := 16.38, [117].Codigo_EAN := '17702161820113', [117].Codigo_QAD := '607020', [117].Codigo_GCO := 607020, [117].Descripcion := 'Aceite Vegetal Torino  Exp.', [117].Cajas_X_Estiba := 48, [117].Codigo_Aceite := 607020, [117].Envase := 17250, [117].Envases_x_Caja := 1, [118].Peso_Real_Estiba := 631.28, [118].Codigo_EAN := '0', [118].Codigo_QAD := '0', [118].Descripcion := '0', [119].Peso_Real_Estiba := 744.8, [119].Codigo_EAN := '0', [119].Codigo_QAD := '0', [119].Descripcion := '0', [120].Peso_Real_Estiba := 827.4, [120].Codigo_EAN := '0', [120].Codigo_QAD := '0', [120].Descripcion := '0', [121].Peso_Real_Estiba := 902.4, [121].Codigo_EAN := '0', [121].Codigo_QAD := '0', [121].Descripcion := '0', [122].Peso_Real_Estiba := 648.0, [122].Codigo_EAN := '0', [122].Codigo_QAD := '0', [122].Descripcion := '0', [123].Peso_Real_Estiba := 869.0, [123].Codigo_EAN := '0', [123].Codigo_QAD := '0', [123].Descripcion := '0',
        [124].Peso_Real_Estiba := 698.4, [124].Codigo_EAN := '0', [124].Codigo_QAD := '0', [124].Descripcion := '0', [125].Peso_Real_Estiba := 746.9, [125].Codigo_EAN := '0', [125].Codigo_QAD := '0', [125].Descripcion := '0', [126].Peso_Real_Estiba := 732.9, [126].Codigo_EAN := '0', [126].Codigo_QAD := '0', [126].Descripcion := '0', [127].Peso_Real_Estiba := 866.5, [127].Codigo_EAN := '0', [127].Codigo_QAD := '0', [127].Descripcion := '0', [128].Peso_Real_Estiba := 691.2, [128].Codigo_EAN := '0', [128].Codigo_QAD := '0', [128].Descripcion := '0', [129].Peso_Real_Estiba := 824.6, [129].Codigo_EAN := '0', [129].Codigo_QAD := '0', [129].Descripcion := '0', [130].Peso_Real_Estiba := 627.12, [130].Codigo_EAN := '0', [130].Codigo_QAD := '0', [130].Descripcion := '0', [131].Peso_Real_Estiba := 733.6, [131].Codigo_EAN := '0', [131].Codigo_QAD := '0', [131].Descripcion := '0', [132].Peso_Real_Estiba := 814.8, [132].Codigo_EAN := '0', [132].Codigo_QAD := '0', [132].Descripcion := '0', [133].Peso_Real_Estiba := 741.3, [133].Codigo_EAN := '0', [133].Codigo_QAD := '0', [133].Descripcion := '0', [134].Peso_Real_Estiba := 741.3, [134].Codigo_EAN := '0', [134].Codigo_QAD := '0', [134].Descripcion := '0', [135].Peso_Real_Estiba := 870.0, [135].Codigo_EAN := '0', [135].Codigo_QAD := '0', [135].Descripcion := '0', [136].Peso_Real_Estiba := 870.0, [136].Codigo_EAN := '0', [136].Codigo_QAD := '0', [136].Descripcion := '0', [137].Peso_Real_Estiba := 693.36, [137].Codigo_EAN := '0', [137].Codigo_QAD := '0', [137].Descripcion := '0', [138].Peso_Real_Estiba := 693.36, [138].Codigo_EAN := '0', [138].Codigo_QAD := '0', [138].Descripcion := '0',
        [139].Peso_Real_Estiba := 820.4, [139].Codigo_EAN := '0', [139].Codigo_QAD := '0', [139].Descripcion := '0', [140].Peso_Real_Estiba := 827.4, [140].Codigo_EAN := '0', [140].Codigo_QAD := '0', [140].Descripcion := '0', [141].Peso_Real_Estiba := 632.32, [141].Codigo_EAN := '0', [141].Codigo_QAD := '0', [141].Descripcion := '0', [142].Peso_Real_Estiba := 742.0, [142].Codigo_EAN := '0', [142].Codigo_QAD := '0', [142].Descripcion := '0', [143].Peso_Real_Estiba := 742.0, [143].Codigo_EAN := '0', [143].Codigo_QAD := '0', [143].Descripcion := '0', [144].Peso_Real_Estiba := 820.4, [144].Codigo_EAN := '0', [144].Codigo_QAD := '0', [144].Descripcion := '0', [145].Peso_Real_Estiba := 820.4, [145].Codigo_EAN := '0', [145].Codigo_QAD := '0', [145].Descripcion := '0', [146].Peso_Real_Estiba := 903.36, [146].Codigo_EAN := '0', [146].Codigo_QAD := '0', [146].Descripcion := '0', [147].Peso_Real_Estiba := 345.4, [147].Codigo_EAN := '0', [147].Codigo_QAD := '0', [147].Descripcion := '0', [148].Peso_Real_Estiba := 633.36, [148].Codigo_EAN := '0', [148].Codigo_QAD := '0', [148].Descripcion := '0', [149].Peso_Real_Estiba := 875.0, [149].Codigo_EAN := '0', [149].Codigo_QAD := '0', [149].Descripcion := '0', [150].Peso_Real_Estiba := 698.4, [150].Codigo_EAN := '0', [150].Codigo_QAD := '0', [150].Descripcion := '0', [151].Peso_Real_Estiba := 816.9, [151].Codigo_EAN := '0', [151].Codigo_QAD := '0', [151].Descripcion := '0', [152].Peso_Real_Estiba := 738.5, [152].Codigo_EAN := '0', [152].Codigo_QAD := '0', [152].Descripcion := '0', [153].Peso_Real_Estiba := 870.0, [153].Codigo_EAN := '0', [153].Codigo_QAD := '0', [153].Descripcion := '0',
        [154].Peso_Real_Estiba := 830.2, [154].Codigo_EAN := '0', [154].Codigo_QAD := '0', [154].Descripcion := '0', [155].Peso_Real_Estiba := 821.1, [155].Codigo_EAN := '0', [155].Codigo_QAD := '0', [155].Descripcion := '0', [156].Peso_Real_Estiba := 743.4, [156].Codigo_EAN := '0', [156].Codigo_QAD := '0', [156].Descripcion := '0', [157].Peso_Real_Estiba := 831.5, [157].Codigo_EAN := '0', [157].Codigo_QAD := '0', [157].Descripcion := '0', [158].Peso_Real_Estiba := 902.88, [158].Codigo_EAN := '0', [158].Codigo_QAD := '0', [158].Descripcion := '0', [159].Peso_Real_Estiba := 691.2, [159].Codigo_EAN := '0', [159].Codigo_QAD := '0', [159].Descripcion := '0', [160].Peso_Real_Estiba := 826.0, [160].Codigo_EAN := '0', [160].Codigo_QAD := '0', [160].Descripcion := '0', [161].Peso_Real_Estiba := 635.44, [161].Codigo_EAN := '0', [161].Codigo_QAD := '0', [161].Descripcion := '0', [162].Peso_Real_Estiba := 746.9, [162].Codigo_EAN := '0', [162].Codigo_QAD := '0', [162].Descripcion := '0', [163].Peso_Real_Estiba := 887.0, [163].Codigo_EAN := '0', [163].Codigo_QAD := '0', [163].Descripcion := '0', [164].Peso_Real_Estiba := 699.84, [164].Codigo_EAN := '0', [164].Codigo_QAD := '0', [164].Descripcion := '0', [165].Peso_Real_Estiba := 833.0, [165].Codigo_EAN := '0', [165].Codigo_QAD := '0', [165].Descripcion := '0', [166].Peso_Real_Estiba := 872.5, [166].Codigo_EAN := '0', [166].Codigo_QAD := '0', [166].Descripcion := '0', [167].Peso_Real_Estiba := 698.4, [167].Codigo_EAN := '0', [167].Codigo_QAD := '0', [167].Descripcion := '0', [168].Peso_Real_Estiba := 747.6, [168].Codigo_EAN := '0', [168].Codigo_QAD := '0', [168].Descripcion := '0',
        [169].Peso_Real_Estiba := 825.3, [169].Codigo_EAN := '0', [169].Codigo_QAD := '0', [169].Descripcion := '0', [170].Peso_Real_Estiba := 880.0, [170].Codigo_EAN := '0', [170].Codigo_QAD := '0', [170].Descripcion := '0', [171].Peso_Real_Estiba := 744.8, [171].Codigo_EAN := '0', [171].Codigo_QAD := '0', [171].Descripcion := '0', [172].Peso_Real_Estiba := 880.0, [172].Codigo_EAN := '0', [172].Codigo_QAD := '0', [172].Descripcion := '0', [173].Peso_Real_Estiba := 739.2, [173].Codigo_EAN := '0', [173].Codigo_QAD := '0', [173].Descripcion := '0', [174].Peso_Real_Estiba := 880.0, [174].Codigo_EAN := '0', [174].Codigo_QAD := '0', [174].Descripcion := '0', [175].Peso_Real_Estiba := 738.5, [175].Codigo_EAN := '0', [175].Codigo_QAD := '0', [175].Descripcion := '0', [176].Peso_Real_Estiba := 875.0, [176].Codigo_EAN := '0', [176].Codigo_QAD := '0', [176].Descripcion := '0', [177].Peso_Real_Estiba := 743.4, [177].Codigo_EAN := '0', [177].Codigo_QAD := '0', [177].Descripcion := '0', [178].Peso_Real_Estiba := 879.0, [178].Codigo_EAN := '0', [178].Codigo_QAD := '0', [178].Descripcion := '0', [179].Peso_Real_Estiba := 703.44, [179].Codigo_EAN := '0', [179].Codigo_QAD := '0', [179].Descripcion := '0', [180].Peso_Real_Estiba := 835.8, [180].Codigo_EAN := '0', [180].Codigo_QAD := '0', [180].Descripcion := '0', [181].Peso_Real_Estiba := 744.8, [181].Codigo_EAN := '0', [181].Codigo_QAD := '0', [181].Descripcion := '0', [182].Peso_Real_Estiba := 905.76, [182].Codigo_EAN := '0', [182].Codigo_QAD := '0', [182].Descripcion := '0', [183].Peso_Real_Estiba := 693.72, [183].Codigo_EAN := '0', [183].Codigo_QAD := '0', [183].Descripcion := '0',
        [184].Peso_Real_Estiba := 880.5, [184].Codigo_EAN := '0', [184].Codigo_QAD := '0', [184].Descripcion := '0', [185].Peso_Real_Estiba := 884.0, [185].Codigo_EAN := '0', [185].Codigo_QAD := '0', [185].Descripcion := '0', [186].Peso_Real_Estiba := 694.44, [186].Codigo_EAN := '0', [186].Codigo_QAD := '0', [186].Descripcion := '0', [187].Peso_Real_Estiba := 928.8, [187].Codigo_EAN := '0', [187].Codigo_QAD := '0', [187].Descripcion := '0', [188].Peso_Real_Estiba := 747.6, [188].Codigo_EAN := '0', [188].Codigo_QAD := '0', [188].Descripcion := '0', [189].Peso_Real_Estiba := 880.0, [189].Codigo_EAN := '0', [189].Codigo_QAD := '0', [189].Descripcion := '0', [190].Peso_Real_Estiba := 698.4, [190].Codigo_EAN := '0', [190].Codigo_QAD := '0', [190].Descripcion := '0', [191].Peso_Real_Estiba := 829.5, [191].Codigo_EAN := '0', [191].Codigo_QAD := '0', [191].Descripcion := '0', [192].Peso_Real_Estiba := 642.72, [192].Codigo_EAN := '0', [192].Codigo_QAD := '0', [192].Descripcion := '0', [193].Peso_Real_Estiba := 743.4, [193].Codigo_EAN := '0', [193].Codigo_QAD := '0', [193].Descripcion := '0', [194].Peso_Real_Estiba := 824.6, [194].Codigo_EAN := '0', [194].Codigo_QAD := '0', [194].Descripcion := '0', [195].Peso_Real_Estiba := 904.32, [195].Codigo_EAN := '0', [195].Codigo_QAD := '0', [195].Descripcion := '0', [196].Peso_Real_Estiba := 648.0, [196].Codigo_EAN := '0', [196].Codigo_QAD := '0', [196].Descripcion := '0', [197].Peso_Real_Estiba := 691.704, [197].Codigo_EAN := '0', [197].Codigo_QAD := '0', [197].Descripcion := '0', [198].Peso_Real_Estiba := 883.2, [198].Codigo_EAN := '0', [198].Codigo_QAD := '0', [198].Descripcion := '0',
        [199].Peso_Real_Estiba := 833.28, [199].Codigo_EAN := '0', [199].Codigo_QAD := '0', [199].Descripcion := '0', [200].Peso_Real_Estiba := 816.9648, [200].Codigo_EAN := '0', [200].Codigo_QAD := '0', [200].Descripcion := '0', [201].Peso_Real_Estiba := 812.64, [201].Codigo_EAN := '0', [201].Codigo_QAD := '0', [201].Descripcion := '0', [202].Peso_Real_Estiba := 907.2, [202].Codigo_EAN := '0', [202].Codigo_QAD := '0', [202].Descripcion := '0', [203].Peso_Real_Estiba := 869.0, [203].Codigo_EAN := '0', [203].Codigo_QAD := '0', [203].Descripcion := '0', [204].Peso_Real_Estiba := 872.0, [204].Codigo_EAN := '0', [204].Codigo_QAD := '0', [204].Descripcion := '0', [205].Peso_Real_Estiba := 870.0, [205].Codigo_EAN := '0', [205].Codigo_QAD := '0', [205].Descripcion := '0', [206].Peso_Real_Estiba := 738.5, [206].Codigo_EAN := '0', [206].Codigo_QAD := '0', [206].Descripcion := '0', [207].Peso_Real_Estiba := 665.0, [207].Codigo_EAN := '0', [207].Codigo_QAD := '0', [207].Descripcion := '0', [208].Peso_Real_Estiba := 617.4, [208].Codigo_EAN := '0', [208].Codigo_QAD := '0', [208].Descripcion := '0', [209].Peso_Real_Estiba := 867.0, [209].Codigo_EAN := '0', [209].Codigo_QAD := '0', [209].Descripcion := '0', [210].Codigo_EAN := '0', [210].Codigo_QAD := '0', [210].Descripcion := '0', [211].Codigo_EAN := '0', [211].Codigo_QAD := '0', [211].Descripcion := '0', [212].Codigo_EAN := '0', [212].Codigo_QAD := '0', [212].Descripcion := '0', [213].Codigo_EAN := '0', [213].Codigo_QAD := '0', [213].Descripcion := '0', [214].Codigo_EAN := '0', [214].Codigo_QAD := '0', [214].Descripcion := '0', [215].Codigo_EAN := '0',
        [215].Codigo_QAD := '0', [215].Descripcion := '0', [216].Codigo_EAN := '0', [216].Codigo_QAD := '0', [216].Descripcion := '0', [217].Codigo_EAN := '0', [217].Codigo_QAD := '0', [217].Descripcion := '0', [218].Codigo_EAN := '0', [218].Codigo_QAD := '0', [218].Descripcion := '0', [219].Codigo_EAN := '0', [219].Codigo_QAD := '0', [219].Descripcion := '0', [220].Codigo_EAN := '0', [220].Codigo_QAD := '0', [220].Descripcion := '0', [221].Codigo_EAN := '0', [221].Codigo_QAD := '0', [221].Descripcion := '0', [222].Codigo_QAD := '0', [222].Descripcion := '0', [223].Codigo_QAD := '0', [223].Descripcion := '0', [224].Codigo_EAN := '0', [224].Codigo_QAD := '0', [224].Descripcion := '0', [225].Codigo_EAN := '0', [225].Codigo_QAD := '0', [225].Descripcion := '0', [226].Codigo_EAN := '0', [226].Codigo_QAD := '0', [226].Descripcion := '0', [227].Codigo_EAN := '0', [227].Codigo_QAD := '0', [227].Descripcion := '0', [228].Codigo_EAN := '0', [228].Codigo_QAD := '0', [228].Descripcion := '0', [229].Codigo_EAN := '0', [229].Codigo_QAD := '0', [229].Descripcion := '0', [230].Codigo_EAN := '0', [230].Codigo_QAD := '0', [230].Descripcion := '0', [231].Codigo_EAN := '0', [231].Codigo_QAD := '0', [231].Descripcion := '0', [232].Codigo_EAN := '0', [232].Codigo_QAD := '0', [232].Descripcion := '0', [233].Codigo_EAN := '0', [233].Codigo_QAD := '0', [233].Descripcion := '0', [234].Codigo_EAN := '0', [234].Codigo_QAD := '0', [234].Descripcion := '0', [235].Codigo_EAN := '0', [235].Codigo_QAD := '0', [235].Descripcion := '0',
        [236].Codigo_EAN := '0', [236].Codigo_QAD := '0', [236].Descripcion := '0', [237].Codigo_EAN := '0', [237].Codigo_QAD := '0', [237].Descripcion := '0', [238].Codigo_EAN := '0', [238].Codigo_QAD := '0', [238].Descripcion := '0', [239].Codigo_EAN := '0', [239].Codigo_QAD := '0', [239].Descripcion := '0', [240].Codigo_EAN := '0', [240].Codigo_QAD := '0', [240].Descripcion := '0', [241].Codigo_EAN := '0', [241].Codigo_QAD := '0', [241].Descripcion := '0', [242].Codigo_EAN := '0', [242].Codigo_QAD := '0', [242].Descripcion := '0', [243].Codigo_EAN := '0', [243].Codigo_QAD := '0', [243].Descripcion := '0', [244].Codigo_EAN := '0', [244].Codigo_QAD := '0', [244].Descripcion := '0', [245].Codigo_EAN := '0', [245].Codigo_QAD := '0', [245].Descripcion := '0', [246].Codigo_EAN := '0', [246].Codigo_QAD := '0', [246].Descripcion := '0', [247].Codigo_EAN := '0', [247].Codigo_QAD := '0', [247].Descripcion := '0', [248].Codigo_EAN := '0', [248].Codigo_QAD := '0', [248].Descripcion := '0', [249].Codigo_EAN := '0', [249].Codigo_QAD := '0', [249].Descripcion := '0', [250].Codigo_EAN := '0', [250].Codigo_QAD := '0', [250].Descripcion := '0', [251].Codigo_EAN := '0', [251].Codigo_QAD := '0', [251].Descripcion := '0', [252].Codigo_EAN := '0', [252].Codigo_QAD := '0', [252].Descripcion := '0', [253].Codigo_EAN := '0', [253].Codigo_QAD := '0', [253].Descripcion := '0', [254].Codigo_EAN := '0', [254].Codigo_QAD := '0', [254].Descripcion := '0', [255].Codigo_EAN := '0', [255].Codigo_QAD := '0', [255].Descripcion := '0',
        [256].Codigo_EAN := '0', [256].Codigo_QAD := '0', [256].Descripcion := '0', [257].Codigo_EAN := '0', [257].Codigo_QAD := '0', [257].Descripcion := '0', [258].Codigo_EAN := '0', [258].Codigo_QAD := '0', [258].Descripcion := '0', [259].Codigo_EAN := '0', [259].Codigo_QAD := '0', [259].Descripcion := '0', [260].Codigo_EAN := '0', [260].Codigo_QAD := '0', [260].Descripcion := '0', [261].Codigo_EAN := '0', [261].Codigo_QAD := '0', [261].Descripcion := '0', [262].Codigo_EAN := '0', [262].Codigo_QAD := '0', [262].Descripcion := '0', [263].Codigo_EAN := '0', [263].Codigo_QAD := '0', [263].Descripcion := '0', [264].Codigo_EAN := '0', [264].Codigo_QAD := '0', [264].Descripcion := '0', [265].Codigo_EAN := '0', [265].Codigo_QAD := '0', [265].Descripcion := '0', [266].Codigo_EAN := '0', [266].Codigo_QAD := '0', [266].Descripcion := '0', [267].Codigo_EAN := '0', [267].Codigo_QAD := '0', [267].Descripcion := '0', [268].Codigo_EAN := '0', [268].Codigo_QAD := '0', [268].Descripcion := '0', [269].Codigo_EAN := '0', [269].Codigo_QAD := '0', [269].Descripcion := '0', [270].Codigo_EAN := '0', [270].Codigo_QAD := '0', [270].Descripcion := '0', [271].Codigo_EAN := '0', [271].Codigo_QAD := '0', [271].Descripcion := '0', [272].Codigo_EAN := '0', [272].Codigo_QAD := '0', [272].Descripcion := '0', [273].Codigo_EAN := '0', [273].Codigo_QAD := '0', [273].Descripcion := '0', [274].Codigo_EAN := '0', [274].Codigo_QAD := '0', [274].Descripcion := '0', [275].Codigo_EAN := '0', [275].Codigo_QAD := '0', [275].Descripcion := '0',
        [276].Codigo_EAN := '0', [276].Codigo_QAD := '0', [276].Descripcion := '0', [277].Codigo_EAN := '0', [277].Codigo_QAD := '0', [277].Descripcion := '0', [278].Codigo_EAN := '0', [278].Codigo_QAD := '0', [278].Descripcion := '0', [279].Codigo_EAN := '0', [279].Codigo_QAD := '0', [279].Descripcion := '0', [280].Codigo_EAN := '0', [280].Codigo_QAD := '0', [280].Descripcion := '0', [281].Codigo_EAN := '0', [281].Codigo_QAD := '0', [281].Descripcion := '0', [282].Codigo_EAN := '0', [282].Codigo_QAD := '0', [282].Descripcion := '0', [283].Codigo_EAN := '0', [283].Codigo_QAD := '0', [283].Descripcion := '0', [284].Codigo_EAN := '0', [284].Codigo_QAD := '0', [284].Descripcion := '0', [285].Codigo_EAN := '0', [285].Codigo_QAD := '0', [285].Descripcion := '0', [286].Codigo_EAN := '0', [286].Codigo_QAD := '0', [286].Descripcion := '0', [287].Codigo_EAN := '0', [287].Codigo_QAD := '0', [287].Descripcion := '0', [288].Codigo_EAN := '0', [288].Codigo_QAD := '0', [288].Descripcion := '0', [289].Codigo_EAN := '0', [289].Codigo_QAD := '0', [289].Descripcion := '0', [290].Codigo_EAN := '0', [290].Codigo_QAD := '0', [290].Descripcion := '0', [291].Codigo_EAN := '0', [291].Codigo_QAD := '0', [291].Descripcion := '0', [292].Codigo_EAN := '0', [292].Codigo_QAD := '0', [292].Descripcion := '0', [293].Codigo_EAN := '0', [293].Codigo_QAD := '0', [293].Descripcion := '0', [294].Codigo_EAN := '0', [294].Codigo_QAD := '0', [294].Descripcion := '0', [295].Codigo_EAN := '0', [295].Codigo_QAD := '0', [295].Descripcion := '0',
        [296].Codigo_EAN := '0', [296].Codigo_QAD := '0', [296].Descripcion := '0', [297].Codigo_EAN := '0', [297].Codigo_QAD := '0', [297].Descripcion := '0', [298].Codigo_EAN := '0', [298].Codigo_QAD := '0', [298].Descripcion := '0', [299].Codigo_EAN := '0', [299].Codigo_QAD := '0', [299].Descripcion := '0');
   Prueba : UDT_COLA[3] := ([0].Fecha.year := 2017, [0].Fecha.Mes := 10, [0].Fecha.Dia := 17, [0].Fecha.Hora := 8, [0].Fecha.Minuto := 37, [0].Fecha.Segundo := 20, [0].Fecha.Milisegundos := 247824, [0].Lote := 290, [0].Operador := 5, [0].Descripcion := 'Vivi Caja 9 x 2000 cm3', [0].EAN14 := '27702179003208', [0].QAD := '7110', [0].Peso_Real := 732.0, [0].Peso_Teorico := 738.0, [0].No_Cajas := 42, [0].Clima := 2, [1].Fecha.year := 2017, [1].Fecha.Mes := 10, [1].Fecha.Dia := 17, [1].Fecha.Hora := 8, [1].Fecha.Minuto := 52, [1].Fecha.Segundo := 44, [1].Fecha.Milisegundos := 604571, [1].Lote := 290, [1].Operador := 5, [1].Descripcion := 'Frescampo Caja 24 x 200 cm3', [1].EAN14 := '67702179095201', [1].QAD := '9520', [1].Peso_Real := 305.0, [1].Peso_Teorico := 304.0, [1].No_Cajas := 62, [1].Clima := 2, [2].Fecha.year := 2017, [2].Fecha.Mes := 10, [2].Fecha.Dia := 17, [2].Fecha.Hora := 10, [2].Fecha.Minuto := 55, [2].Fecha.Segundo := 12, [2].Fecha.Milisegundos := 443803, [2].Lote := 290, [2].Descripcion := ' Oriental Caja 6 x 3000 cm3', [2].EAN14 := '17702161303159', [2].QAD := '5050', [2].Peso_Teorico := 880.0, [2].No_Cajas := 50, [2].Clima := 2);
   Prueba_Bit : BOOL;
   Prueba_Index : DINT;
   Prueba_X : BOOL;
   PV_Datos_Mal_Bidones : BOOL;
   PV_Datos_Mal_Elmar : BOOL;
   PV_Datos_Mal_Fogg1 : BOOL;
   PV_Datos_Mal_Fogg2 : BOOL;
   PV_Datos_Mal_Karat : BOOL;
   PV_Datos_Malos_Elmar : BOOL;
   PV_Datos_Malos_Fogg2 : BOOL;
   PV_Datos_Malos_Karat : BOOL;
   PV_Datos_Pesaje_Bidones : BOOL;
   PV_Datos_Pesaje_Elmar : BOOL;
   PV_Datos_Pesaje_Fogg1 : BOOL;
   PV_Datos_Pesaje_Fogg2 : BOOL;
   PV_Datos_Pesaje_Karat : BOOL;
   QAD_1 : STRING := '605990';
   QAD_2 : STRING := '600620';
   QAD_3 : STRING := '605990';
   QAD_4 : STRING := '607020';
   QAD_Aux : DINT;
   QAD_Aux_Scanner : STRING;
   QAD_Auxiliar_Est1 : STRING := '605990';
   QAD_Auxiliar_Est2 : STRING := '600620';
   QAD_Auxiliar_Est3 : STRING := '605990';
   QAD_Auxiliar_Est4 : STRING := '607020';
   Report_Con1 : BOOL := 1;
   Reporte_Dia_Lach : BOOL;
   Reporte_Dia_Timer : TIMER := (PRE := 5000);
   Reporte_Scanner : BOOL;
   Revisa_Pesaje_1 : BOOL;
   Revisar_Peso_Teorico_1 : BOOL;
   Revision_Peso_1 : Revision_Peso := (Date.year := 2017, Date.Mes := 10, Date.Dia := 6, Date.Hora := 10, Date.Minuto := 22, Date.Segundo := 2, Date.Milisegundos := 677509, Peso_Real := 639.0, Peso_Teorico := 225.0);
   Revision_Peso_2 : Revision_Peso;
   Sin_Codigo : UDT_QAD;
   Sin_Codigo_21 : STRING;
   Slash : STRING := '/';
   Station1_Tare_OK : BOOL := 1;
   Station2_Tare_OK : BOOL := 1;
   Station3_Tare_OK : BOOL := 1;
   Station4_Tare_OK : BOOL := 1;
   SYSTEM_ALARMS : DINT[10] := ([0] := 16777216);
   SYSTEM_STATUS_COMPLETE : BOOL := 1;
   Tara_1 : DINT := 2;
   Tara_2 : DINT := 16777218;
   Tara_3 : DINT := 33554434;
   Tara_4 : DINT := 50331650;
   Tara_Fecha_Estacion_1 : Hora_y_Fecha := (year := 2020, Mes := 11, Dia := 7, Hora := 12, Minuto := 2, Segundo := 32, Milisegundos := 549887);
   Tara_Fecha_Estacion_2 : Hora_y_Fecha := (year := 2021, Mes := 5, Dia := 28, Hora := 14, Minuto := 38, Segundo := 42, Milisegundos := 7920);
   Tara_Fecha_Estacion_3 : Hora_y_Fecha := (year := 2021, Mes := 5, Dia := 28, Hora := 16, Minuto := 13, Segundo := 48, Milisegundos := 39475);
   Tara_Fecha_Estacion_4 : Hora_y_Fecha := (year := 2021, Mes := 5, Dia := 28, Hora := 14, Minuto := 43, Segundo := 13, Milisegundos := 444987);
   Tare_Station_1_Read : DINT := 33554432;
   Tare_Station_1_Write : DINT := 2;
   Tare_Station_2_Write : DINT := 16777218;
   Tare_Station_3_Write : DINT := 33554434;
   Tare_Station_4_Write : DINT := 50331650;
   time_new : TIMER := (PRE := 3000);
   Timer_Datos_Bidones : TIMER := (PRE := 50000);
   Timer_Print_1 : TIMER := (PRE := 2000);
   Timer_Print_2 : TIMER := (PRE := 2000);
   Timer_Print_3 : TIMER;
   Timer_Reporte_Scanner : TIMER := (PRE := 5000);
   TRES : SINT := 3;
   try : BOOL;
   U_Fecha_Bidones : Hora_y_Fecha := (year := 2020, Mes := 7, Dia := 28, Hora := 12, Minuto := 39, Segundo := 29, Milisegundos := 53247);
   U_Fecha_Elmar : Hora_y_Fecha := (year := 2020, Mes := 5, Dia := 21, Hora := 17, Minuto := 3, Segundo := 26, Milisegundos := 553850);
   U_Fecha_Fogg1 : Hora_y_Fecha := (year := 2020, Mes := 3, Dia := 12, Hora := 9, Minuto := 54, Segundo := 23, Milisegundos := 724385);
   U_Fecha_Fogg2 : Hora_y_Fecha := (year := 2020, Mes := 5, Dia := 21, Hora := 17, Minuto := 3, Segundo := 43, Milisegundos := 873934);
   U_Fecha_Karat : Hora_y_Fecha;
   Un_Espacio : STRING := ' ';
   UNO : SINT := 1;
   Velocidad_Modo_Forzado : BOOL;
   WPM1_Heartbeat : DINT := 4;
   WPM1_Heartbeat_Error : BOOL := 1;
   WPM1_Status : WPM_Status;
   WPM2_Heartbeat : DINT := 1;
   WPM2_Heartbeat_Error : BOOL := 1;
   WPM2_Status : WPM_Status;
   WPM3_Heartbeat : DINT := 7;
   WPM3_Heartbeat_Error : BOOL := 1;
   WPM3_Status : WPM_Status;
   WPM4_Heartbeat : DINT := 1;
   WPM4_Heartbeat_Error : BOOL := 1;
   WPM4_Status : WPM_Status;
   WPM_1_Selected : DINT;
   WPM_1_Status_Aux : DINT;
   WPM_2_COUNT_ANTERIOR : DINT := 1;
   WPM_2_Selected : DINT := 1;
   WPM_2_Status_Aux : DINT;
   WPM_3_Selected : DINT := 2;
   WPM_3_Status_Aux : DINT;
   WPM_4_Selected : DINT := 3;
   WPM_4_Status_Aux : DINT;
   Zero : DINT;
END_VAR
